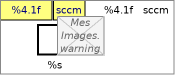
VISUALIZATION VISU_MFC_ANA  // 175x75
VAR_IN_OUT
	m_Input_MACHINE:	BLOCK_MODE_MARCHE_V2_0;
	m_Input_MASSFLOW:	BLOCK_MFC_ANA2;
	m_Input_LIGNE_GAZ:	BLOCK_LIGNE_GAZ;
END_VAR
    Rectangle (37,24 34x31)
    RoundedRectangle (0,0 52x20), "%4.1f", text variable: m_Input_MASSFLOW.PRM_Flow, invisible if: (m_Input_MACHINE.STATE_Manu) <> 0
    Rectangle (90,0 49x20), "%4.1f", text variable: m_Input_MASSFLOW.STATE_Flow
    RoundedRectangle (53,0 32x20), "sccm"
    Rectangle (140,0 35x20), "sccm"
    Rectangle (35,55 40x20), "%s", text variable: m_Input_MASSFLOW.MNEMO
    RoundedRectangle (0,0 52x20), "%4.1f", text variable: m_Input_LIGNE_GAZ.PRM_Flow, invisible if: NOT m_Input_MACHINE.STATE_Manu, input disabled if: NOT m_Input_MACHINE.STATE_Manu OR NOT PRG_User.ACTU_USER.MAINTENANCE
        OnMouseDown: write the text variable via VisuDialogs.Numpad, min 0, max m_Input_MASSFLOW.CONF_Util_Max_Flow
    Polyline (53,32)
    Polyline (61,39)
    Rectangle (55,39 16x18), "D"
    Image (57,16 47x39), invisible if: NOT m_Input_MASSFLOW.STATE_NOK, image: MesImages.warning
END_VISUALIZATION

(* stored: Version 1.1.0.1, ProductVersion 3.1.4024.10
   Visu VISU_MFC_ANA: Id {fd0d4ddd-433d-47dc-a444-0f51f0875511} *)
